Fanuc KAREL source: kb00136.KL

-- PROVISIONAL review KL for V770-1; original PC SHA256 88b4d68a60dc970c81b480326af3bea2f212ccc863be82456dd54924333af1ab
-- Incomplete behavior may be omitted. Consult companion uncertainty JSON. Do not deploy.
PROGRAM KB00136
%NOLOCKGROUP
BEGIN
  -- UNRESOLVED_PC offsets 5-14; opcodes 3F,75
  -- UNRESOLVED_PC offsets 19-26; opcodes 9D,23
  -- UNRESOLVED_PC offsets 31-38; opcodes 9D,23
  -- UNRESOLVED_PC offsets 43-67; opcodes 27,22,2A,22,22,31
  -- UNRESOLVED_PC offsets 72-76; opcodes 7F
END KB00136
